Fanuc KAREL source: worntmrot.kl

PROGRAM worntmrot
%NOLOCKGROUP
VAR
  p : POSITION
  q : POSITION
  i : INTEGER
  r : REAL
BEGIN
  WITH $ORNT_MROT = TRUE MOVE TO p
END worntmrot
